// TIA Portal V20 export
FUNCTION_BLOCK "FB_ReadWrite_GUDs"   // FB1200, SCL
{ S7_Optimized_Access := 'TRUE' }
// stored: AutoNumber false, MemoryReserve 100, SetENOAutomatically false
   VAR
      sStart_rd { ExternalAccessible := 'False'; ExternalVisible := 'False'; ExternalWritable := 'False'} : Bool;
      sNCK_channel { ExternalAccessible := 'False'; ExternalVisible := 'False'; ExternalWritable := 'False'} : Byte;   // 0:GUD NCK, 1:GUD Chan1, 2:GUD Chan2 etc...
      sType { ExternalAccessible := 'False'; ExternalVisible := 'False'; ExternalWritable := 'False'} : Int;   // 0:Bool, 1:Int, 2:DWord, 3:Real, 4:String
      sName { ExternalAccessible := 'False'; ExternalVisible := 'False'; ExternalWritable := 'False'} : String;   // GUD Name
      sIndex1 { ExternalAccessible := 'False'; ExternalVisible := 'False'; ExternalWritable := 'False'} : Int;
      sindex2 { ExternalAccessible := 'False'; ExternalVisible := 'False'; ExternalWritable := 'False'} : Int;
      sToken_GUD { ExternalAccessible := 'False'; ExternalVisible := 'False'; ExternalWritable := 'False'} : "UDT_Token_GUD";
      sValue_bit { ExternalAccessible := 'False'; ExternalVisible := 'False'; ExternalWritable := 'False'} : Bool;
      sValue_int { ExternalAccessible := 'False'; ExternalVisible := 'False'; ExternalWritable := 'False'} : Int;
      sValue_double { ExternalAccessible := 'False'; ExternalVisible := 'False'; ExternalWritable := 'False'} : DWord;
      sValue_real { ExternalAccessible := 'False'; ExternalVisible := 'False'; ExternalWritable := 'False'} : Real;
      sValue_String { ExternalAccessible := 'False'; ExternalVisible := 'False'; ExternalWritable := 'False'} : String;
      sStatus_rd { ExternalAccessible := 'False'; ExternalVisible := 'False'; ExternalWritable := 'False'} : Word;
      sRead_done { ExternalAccessible := 'False'; ExternalVisible := 'False'; ExternalWritable := 'False'} : Bool;
      sRead_done_Mem { ExternalAccessible := 'False'; ExternalVisible := 'False'; ExternalWritable := 'False'} : Bool;
      sStart_wr { ExternalAccessible := 'False'; ExternalVisible := 'False'; ExternalWritable := 'False'} : Bool;
      sNumVar_wr { ExternalAccessible := 'False'; ExternalVisible := 'False'; ExternalWritable := 'False'} : Int := 1;
      sAddr_wr { ExternalAccessible := 'False'; ExternalVisible := 'False'; ExternalWritable := 'False'} : Array[0..7] of "UDT_Token_GUD";
      sColumn_wr { ExternalAccessible := 'False'; ExternalVisible := 'False'; ExternalWritable := 'False'} : Array[0..7] of Word;
      sLine_wr { ExternalAccessible := 'False'; ExternalVisible := 'False'; ExternalWritable := 'False'} : Array[0..7] of Word;
      sStatus_wr { ExternalAccessible := 'False'; ExternalVisible := 'False'; ExternalWritable := 'False'} : Word;
      sWrite_done { ExternalAccessible := 'False'; ExternalVisible := 'False'; ExternalWritable := 'False'} : Bool;
      sWriteVal_bit { ExternalAccessible := 'False'; ExternalVisible := 'False'; ExternalWritable := 'False'} : Array[0..7] of Bool;
      sWriteVal_int { ExternalAccessible := 'False'; ExternalVisible := 'False'; ExternalWritable := 'False'} : Array[0..7] of Int;
      sWriteVal_double { ExternalAccessible := 'False'; ExternalVisible := 'False'; ExternalWritable := 'False'} : Array[0..7] of DWord;
      sWriteVal_Real { ExternalAccessible := 'False'; ExternalVisible := 'False'; ExternalWritable := 'False'} : Array[0..7] of DWord;
      sWriteVal_String { ExternalAccessible := 'False'; ExternalVisible := 'False'; ExternalWritable := 'False'} : Array[0..7] of String;
      sLBP_ReadGUD_Instance { ExternalAccessible := 'False'; ExternalVisible := 'False'; ExternalWritable := 'False'} : "LBP_ReadGUD";
      sLBP_WriteGUD_Instance { ExternalAccessible := 'False'; ExternalVisible := 'False'; ExternalWritable := 'False'} : "LBP_WriteVar";
   END_VAR
   VAR_TEMP
      tArea : Byte;
      tUnit : Byte;
      tError : Bool;
      tStatus : Word;
      tLoop_I : Int;
   END_VAR
   // sColumn_wr[0..7] := 16#1;
   // sLine_wr[0..7] := 16#1;
BEGIN
   REGION Reading
       IF #sNCK_channel = 0 THEN
           #tArea := 0;
           #tUnit := 1;
       ELSE
           #tArea := 2;
           #tUnit := #sNCK_channel;
       END_IF;

       CASE #sType OF
           0:
               #sLBP_ReadGUD_Instance(Req := #sStart_rd,
                                     Addr := #sName,
                                     Area := #tArea,
                                     Unit := #tUnit,
                                     Index1 := #sIndex1,
                                     Index2 := #sindex2,
                                     CnvtToken := TRUE,
                                     VarToken := #sToken_GUD,
                                     Error => #tError,
                                     Done => #sRead_done,
                                     State => #tStatus,
                                     RD := #sValue_bit);
           1:
               #sLBP_ReadGUD_Instance(Req := #sStart_rd,
                                     Addr := #sName,
                                     Area := #tArea,
                                     Unit := #tUnit,
                                     Index1 := #sIndex1,
                                     Index2 := #sindex2,
                                     CnvtToken := TRUE,
                                     VarToken := #sToken_GUD,
                                     Error => #tError,
                                     Done => #sRead_done,
                                     State => #tStatus,
                                     RD := #sValue_int);

           2:
               #sLBP_ReadGUD_Instance(Req := #sStart_rd,
                                     Addr := #sName,
                                     Area := #tArea,
                                     Unit := #tUnit,
                                     Index1 := #sIndex1,
                                     Index2 := #sindex2,
                                     CnvtToken := TRUE,
                                     VarToken := #sToken_GUD,
                                     Error => #tError,
                                     Done => #sRead_done,
                                     State => #tStatus,
                                     RD := #sValue_double);

           3:
               #sLBP_ReadGUD_Instance(Req := #sStart_rd,
                                     Addr := #sName,
                                     Area := #tArea,
                                     Unit := #tUnit,
                                     Index1 := #sIndex1,
                                     Index2 := #sindex2,
                                     CnvtToken := TRUE,
                                     VarToken := #sToken_GUD,
                                     Error => #tError,
                                     Done => #sRead_done,
                                     State => #tStatus,
                                     RD := #sValue_real);

           4:
               #sLBP_ReadGUD_Instance(Req := #sStart_rd,
                                     Addr := #sName,
                                     Area := #tArea,
                                     Unit := #tUnit,
                                     Index1 := #sIndex1,
                                     Index2 := #sindex2,
                                     CnvtToken := TRUE,
                                     VarToken := #sToken_GUD,
                                     Error => #tError,
                                     Done => #sRead_done,
                                     State => #tStatus,
                                     RD := #sValue_String);


       END_CASE;

       IF #sRead_done OR #tError THEN
           #sRead_done := TRUE;
           #sStatus_rd := #tStatus;
           #sStart_rd := FALSE;
       END_IF;
       IF #sRead_done AND NOT #sRead_done_Mem THEN
           FOR #tLoop_I := 1 TO 8 DO
               IF #tLoop_I <= #sNumVar_wr THEN
                 #sAddr_wr[#tLoop_I - 1] := #sToken_GUD;
               END_IF;
           END_FOR;
           #sRead_done_Mem := TRUE;
       END_IF;

   END_REGION


   REGION Writing

       CASE #sType OF
           0:
               #sLBP_WriteGUD_Instance(Req := #sStart_wr AND #sRead_done_Mem,
                                      NumVar := #sNumVar_wr,
                                      Addr1 := #sAddr_wr[0],
                                      Line1 := #sLine_wr[0],
                                      Column1 := #sColumn_wr[0],
                                      Addr2 := #sAddr_wr[1],
                                      Line2 := #sLine_wr[1],
                                      Column2 := #sColumn_wr[1],
                                      Addr3 := #sAddr_wr[2],
                                      Line3 := #sLine_wr[2],
                                      Column3 := #sColumn_wr[2],
                                      Addr4 := #sAddr_wr[3],
                                      Line4 := #sLine_wr[3],
                                      Column4 := #sColumn_wr[3],
                                      Addr5 := #sAddr_wr[4],
                                      Line5 := #sLine_wr[4],
                                      Column5 := #sColumn_wr[4],
                                      Addr6 := #sAddr_wr[5],
                                      Line6 := #sLine_wr[5],
                                      Column6 := #sColumn_wr[5],
                                      Addr7 := #sAddr_wr[6],
                                      Line7 := #sLine_wr[6],
                                      Column7 := #sColumn_wr[6],
                                      Addr8 := #sAddr_wr[7],
                                      Line8 := #sLine_wr[7],
                                      Column8 := #sColumn_wr[7],
                                      Error => #tError,
                                      Done => #sWrite_done,
                                      State => #tStatus,
                                      SD1 := #sWriteVal_bit[0],
                                      SD2 := #sWriteVal_bit[1],
                                      SD3 := #sWriteVal_bit[2],
                                      SD4 := #sWriteVal_bit[3],
                                      SD5 := #sWriteVal_bit[4],
                                      SD6 := #sWriteVal_bit[5],
                                      SD7 := #sWriteVal_bit[6],
                                      SD8 := #sWriteVal_bit[7]);
           1:
               #sLBP_WriteGUD_Instance(Req := #sStart_wr AND #sRead_done_Mem,
                                      NumVar := #sNumVar_wr,
                                      Addr1 := #sAddr_wr[0],
                                      Line1 := #sLine_wr[0],
                                      Column1 := #sColumn_wr[0],
                                      Addr2 := #sAddr_wr[1],
                                      Line2 := #sLine_wr[1],
                                      Column2 := #sColumn_wr[1],
                                      Addr3 := #sAddr_wr[2],
                                      Line3 := #sLine_wr[2],
                                      Column3 := #sColumn_wr[2],
                                      Addr4 := #sAddr_wr[3],
                                      Line4 := #sLine_wr[3],
                                      Column4 := #sColumn_wr[3],
                                      Addr5 := #sAddr_wr[4],
                                      Line5 := #sLine_wr[4],
                                      Column5 := #sColumn_wr[4],
                                      Addr6 := #sAddr_wr[5],
                                      Line6 := #sLine_wr[5],
                                      Column6 := #sColumn_wr[5],
                                      Addr7 := #sAddr_wr[6],
                                      Line7 := #sLine_wr[6],
                                      Column7 := #sColumn_wr[6],
                                      Addr8 := #sAddr_wr[7],
                                      Line8 := #sLine_wr[7],
                                      Column8 := #sColumn_wr[7],
                                      Error => #tError,
                                      Done => #sWrite_done,
                                      State => #tStatus,
                                      SD1 := #sWriteVal_int[0],
                                      SD2 := #sWriteVal_int[1],
                                      SD3 := #sWriteVal_int[2],
                                      SD4 := #sWriteVal_int[3],
                                      SD5 := #sWriteVal_int[4],
                                      SD6 := #sWriteVal_int[5],
                                      SD7 := #sWriteVal_int[6],
                                      SD8 := #sWriteVal_int[7]);

           2:
               #sLBP_WriteGUD_Instance(Req := #sStart_wr AND #sRead_done_Mem,
                                      NumVar := #sNumVar_wr,
                                      Addr1 := #sAddr_wr[0],
                                      Line1 := #sLine_wr[0],
                                      Column1 := #sColumn_wr[0],
                                      Addr2 := #sAddr_wr[1],
                                      Line2 := #sLine_wr[1],
                                      Column2 := #sColumn_wr[1],
                                      Addr3 := #sAddr_wr[2],
                                      Line3 := #sLine_wr[2],
                                      Column3 := #sColumn_wr[2],
                                      Addr4 := #sAddr_wr[3],
                                      Line4 := #sLine_wr[3],
                                      Column4 := #sColumn_wr[3],
                                      Addr5 := #sAddr_wr[4],
                                      Line5 := #sLine_wr[4],
                                      Column5 := #sColumn_wr[4],
                                      Addr6 := #sAddr_wr[5],
                                      Line6 := #sLine_wr[5],
                                      Column6 := #sColumn_wr[5],
                                      Addr7 := #sAddr_wr[6],
                                      Line7 := #sLine_wr[6],
                                      Column7 := #sColumn_wr[6],
                                      Addr8 := #sAddr_wr[7],
                                      Line8 := #sLine_wr[7],
                                      Column8 := #sColumn_wr[7],
                                      Error => #tError,
                                      Done => #sWrite_done,
                                      State => #tStatus,
                                      SD1 := #sWriteVal_double[0],
                                      SD2 := #sWriteVal_double[1],
                                      SD3 := #sWriteVal_double[2],
                                      SD4 := #sWriteVal_double[3],
                                      SD5 := #sWriteVal_double[4],
                                      SD6 := #sWriteVal_double[5],
                                      SD7 := #sWriteVal_double[6],
                                      SD8 := #sWriteVal_double[7]);

           3:
               #sLBP_WriteGUD_Instance(Req := #sStart_wr AND #sRead_done_Mem,
                                      NumVar := #sNumVar_wr,
                                      Addr1 := #sAddr_wr[0],
                                      Line1 := #sLine_wr[0],
                                      Column1 := #sColumn_wr[0],
                                      Addr2 := #sAddr_wr[1],
                                      Line2 := #sLine_wr[1],
                                      Column2 := #sColumn_wr[1],
                                      Addr3 := #sAddr_wr[2],
                                      Line3 := #sLine_wr[2],
                                      Column3 := #sColumn_wr[2],
                                      Addr4 := #sAddr_wr[3],
                                      Line4 := #sLine_wr[3],
                                      Column4 := #sColumn_wr[3],
                                      Addr5 := #sAddr_wr[4],
                                      Line5 := #sLine_wr[4],
                                      Column5 := #sColumn_wr[4],
                                      Addr6 := #sAddr_wr[5],
                                      Line6 := #sLine_wr[5],
                                      Column6 := #sColumn_wr[5],
                                      Addr7 := #sAddr_wr[6],
                                      Line7 := #sLine_wr[6],
                                      Column7 := #sColumn_wr[6],
                                      Addr8 := #sAddr_wr[7],
                                      Line8 := #sLine_wr[7],
                                      Column8 := #sColumn_wr[7],
                                      Error => #tError,
                                      Done => #sWrite_done,
                                      State => #tStatus,
                                      SD1 := #sWriteVal_Real[0],
                                      SD2 := #sWriteVal_Real[1],
                                      SD3 := #sWriteVal_Real[2],
                                      SD4 := #sWriteVal_Real[3],
                                      SD5 := #sWriteVal_Real[4],
                                      SD6 := #sWriteVal_Real[5],
                                      SD7 := #sWriteVal_Real[6],
                                      SD8 := #sWriteVal_Real[7]);

           4:
               #sLBP_WriteGUD_Instance(Req := #sStart_wr AND #sRead_done_Mem,
                                      NumVar := #sNumVar_wr,
                                      Addr1 := #sAddr_wr[0],
                                      Line1 := #sLine_wr[0],
                                      Column1 := #sColumn_wr[0],
                                      Addr2 := #sAddr_wr[1],
                                      Line2 := #sLine_wr[1],
                                      Column2 := #sColumn_wr[1],
                                      Addr3 := #sAddr_wr[2],
                                      Line3 := #sLine_wr[2],
                                      Column3 := #sColumn_wr[2],
                                      Addr4 := #sAddr_wr[3],
                                      Line4 := #sLine_wr[3],
                                      Column4 := #sColumn_wr[3],
                                      Addr5 := #sAddr_wr[4],
                                      Line5 := #sLine_wr[4],
                                      Column5 := #sColumn_wr[4],
                                      Addr6 := #sAddr_wr[5],
                                      Line6 := #sLine_wr[5],
                                      Column6 := #sColumn_wr[5],
                                      Addr7 := #sAddr_wr[6],
                                      Line7 := #sLine_wr[6],
                                      Column7 := #sColumn_wr[6],
                                      Addr8 := #sAddr_wr[7],
                                      Line8 := #sLine_wr[7],
                                      Column8 := #sColumn_wr[7],
                                      Error => #tError,
                                      Done => #sWrite_done,
                                      State => #tStatus,
                                      SD1 := #sWriteVal_String[0],
                                      SD2 := #sWriteVal_String[1],
                                      SD3 := #sWriteVal_String[2],
                                      SD4 := #sWriteVal_String[3],
                                      SD5 := #sWriteVal_String[4],
                                      SD6 := #sWriteVal_String[5],
                                      SD7 := #sWriteVal_String[6],
                                      SD8 := #sWriteVal_String[7]);
       END_CASE;

       IF #sWrite_done OR #tError THEN
           #sWrite_done := TRUE;
           #sStatus_wr := #tStatus;
           #sStart_wr := FALSE;
       END_IF;


   END_REGION
END_FUNCTION_BLOCK
